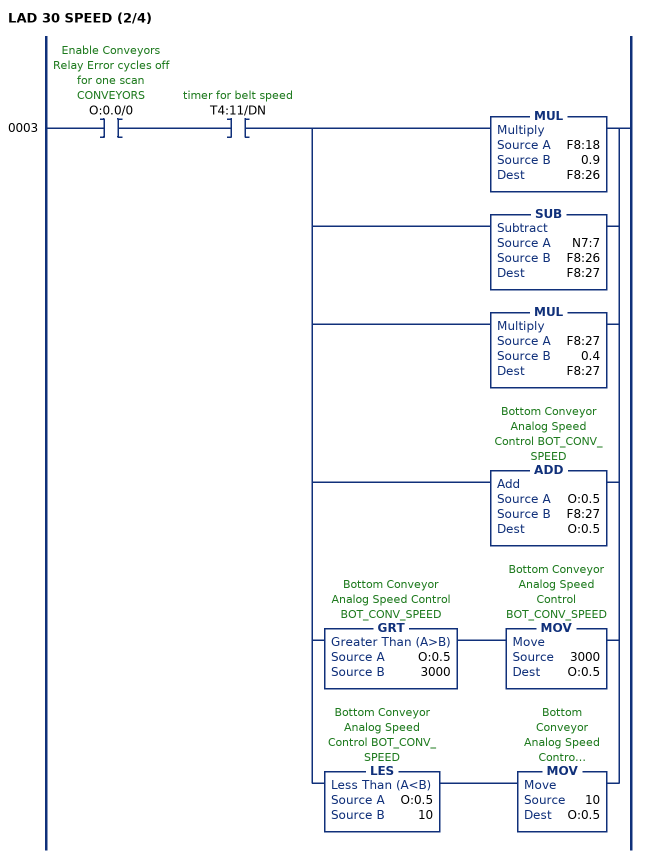
% Rung: 3 %
SOR XIC O:0.0/0 XIC T4:11/DN BST MUL F8:18 0.9 F8:26 NXB SUB N7:7 F8:26 F8:27 NXB MUL F8:27 0.4 F8:27 NXB ADD O:0.5 F8:27 O:0.5 NXB GRT O:0.5 3000 MOV 3000 O:0.5 NXB LES O:0.5 10 MOV 10 O:0.5 BND EOR
%   O:0.0/0  CONVEYORS  "Enable Conveyors Relay Error cycles off for one scan" %
%   T4:11  "timer for belt speed" %
%   F8:18  "top belt speed average in pulses per 100ms" %
%   N7:7  "Top Conv Speed" %
%   O:0.5  BOT_CONV_SPEED  "Bottom Conveyor Analog Speed Control" %

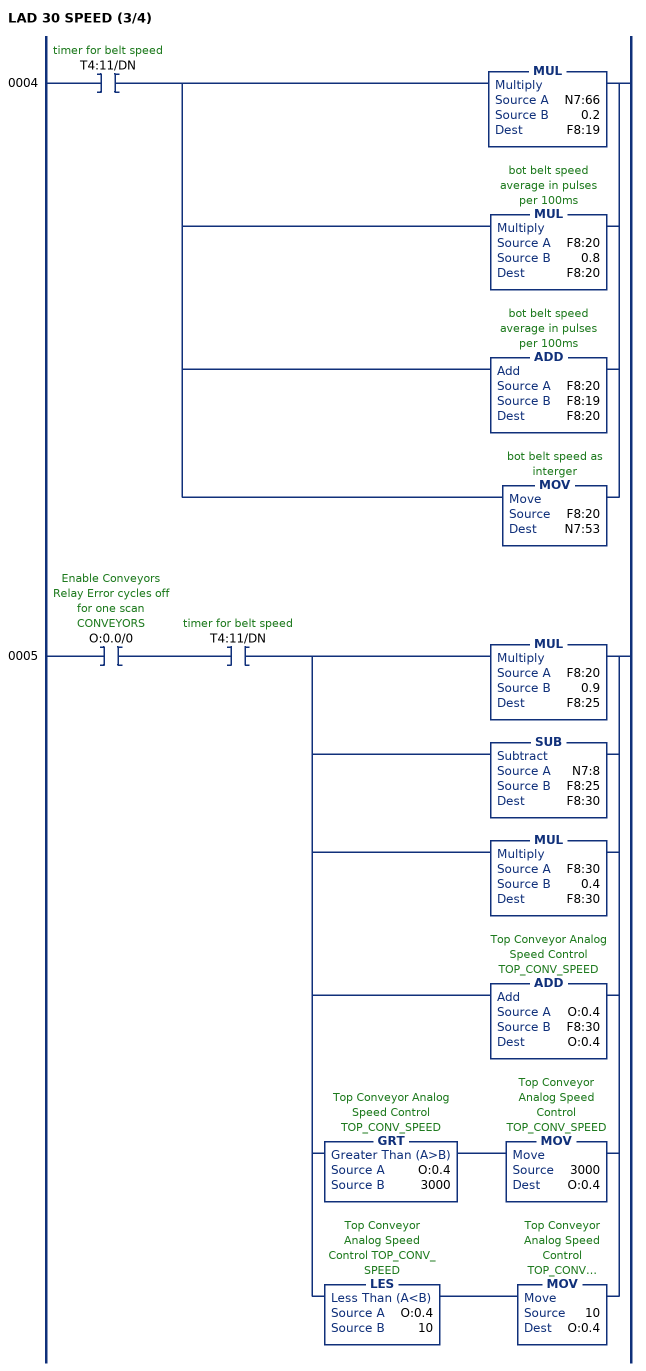
% Rung: 4 %
SOR XIC T4:11/DN BST MUL N7:66 0.2 F8:19 NXB MUL F8:20 0.8 F8:20 NXB ADD F8:20 F8:19 F8:20 NXB MOV F8:20 N7:53 BND EOR
%   T4:11  "timer for belt speed" %
%   N7:66  "pps bottom belt" %
%   F8:20  "bot belt speed average in pulses per 100ms" %
%   N7:53  "bot belt speed as interger" %
% Rung: 5 %
SOR XIC O:0.0/0 XIC T4:11/DN BST MUL F8:20 0.9 F8:25 NXB SUB N7:8 F8:25 F8:30 NXB MUL F8:30 0.4 F8:30 NXB ADD O:0.4 F8:30 O:0.4 NXB GRT O:0.4 3000 MOV 3000 O:0.4 NXB LES O:0.4 10 MOV 10 O:0.4 BND EOR
%   O:0.0/0  CONVEYORS  "Enable Conveyors Relay Error cycles off for one scan" %
%   T4:11  "timer for belt speed" %
%   F8:20  "bot belt speed average in pulses per 100ms" %
%   N7:8  "Bottom Conveyor Speed" %
%   O:0.4  TOP_CONV_SPEED  "Top Conveyor Analog Speed Control" %

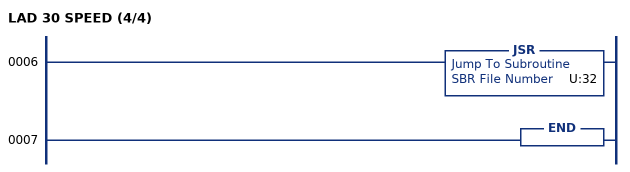
% Rung: 6 %
SOR JSR U:32 EOR
% Rung: 7 %
SOR END EOR

LADDER 32 "BOXER"
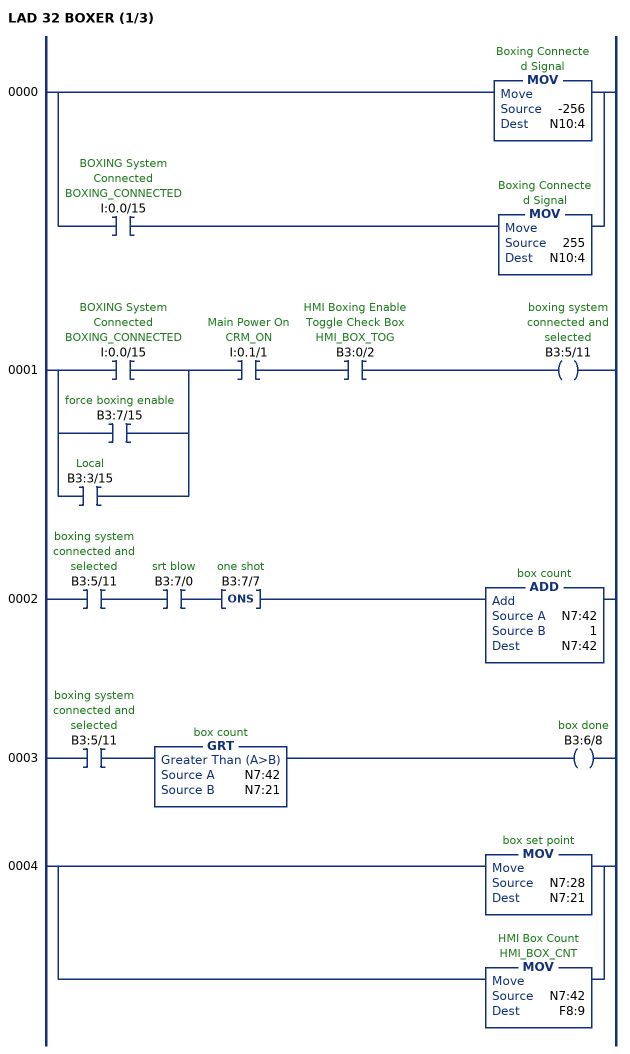
% Rung: 0 %
SOR BST MOV -256 N10:4 NXB XIC I:0.0/15 MOV 255 N10:4 BND EOR
%   N10:4  "Boxing Connected Signal" %
%   I:0.0/15  BOXING_CONNECTED  "BOXING System Connected" %
% Rung: 1 %
SOR BST XIC I:0.0/15 NXB XIC B3:7/15 NXB XIC B3:3/15 BND XIC I:0.1/1 XIC B3:0/2 OTE B3:5/11 EOR
%   I:0.0/15  BOXING_CONNECTED  "BOXING System Connected" %
%   B3:7/15  "force boxing enable" %
%   B3:3/15  "Local" %
%   I:0.1/1  CRM_ON  "Main Power On" %
%   B3:0/2  HMI_BOX_TOG  "HMI Boxing Enable Toggle Check Box" %
%   B3:5/11  "boxing system connected and selected" %
% Rung: 2 %
SOR XIC B3:5/11 XIC B3:7/0 ONS B3:7/7 ADD N7:42 1 N7:42 EOR
%   B3:5/11  "boxing system connected and selected" %
%   B3:7/0  "srt blow" %
%   B3:7/7  "one shot" %
%   N7:42  "box count" %
% Rung: 3 %
SOR XIC B3:5/11 GRT N7:42 N7:21 OTE B3:6/8 EOR
%   B3:5/11  "boxing system connected and selected" %
%   N7:42  "box count" %
%   N7:21  "box set point" %
%   B3:6/8  "box done" %
% Rung: 4 %
SOR BST MOV N7:28 N7:21 NXB MOV N7:42 F8:9 BND EOR
%   N7:28  "box count limit" %
%   N7:21  "box set point" %
%   N7:42  "box count" %
%   F8:9  HMI_BOX_CNT  "HMI Box Count" %

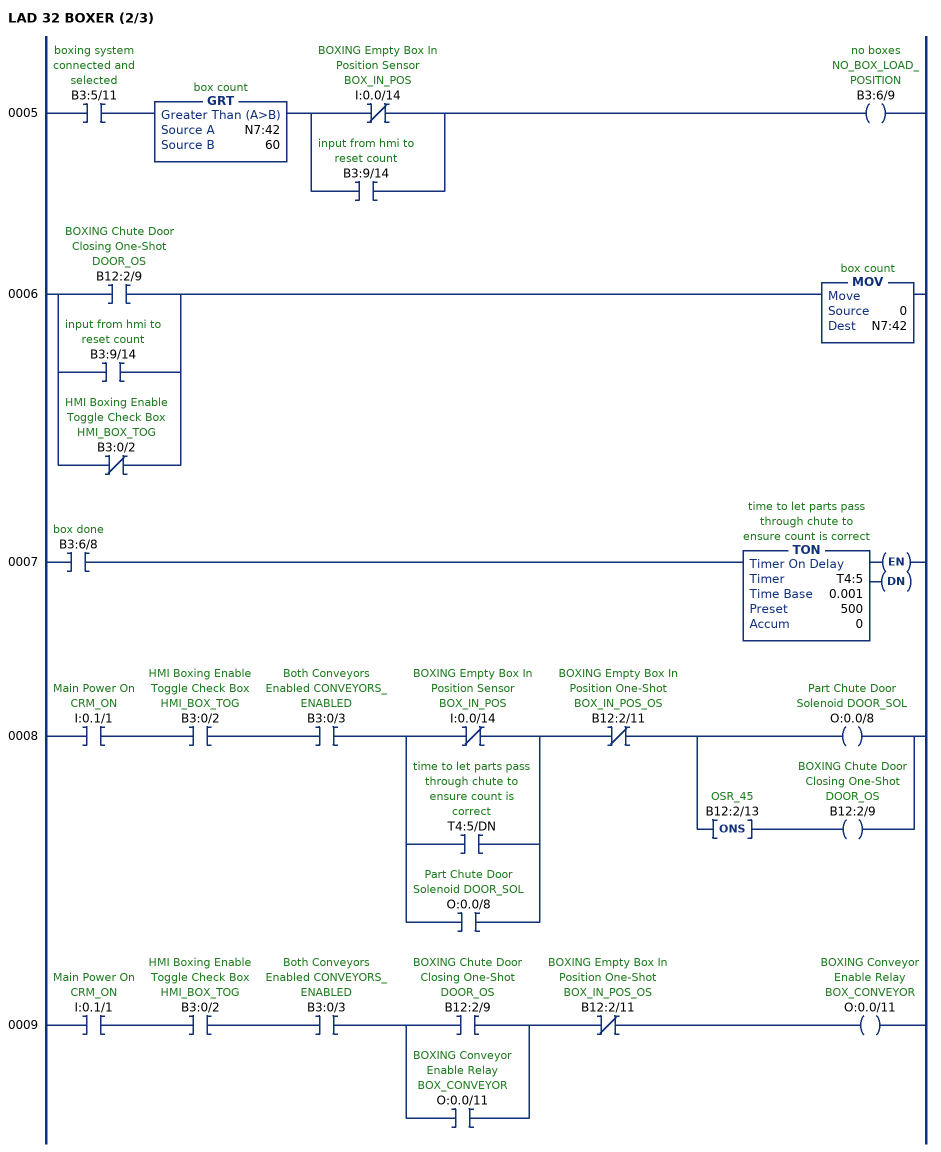
% Rung: 5 %
SOR XIC B3:5/11 GRT N7:42 60 BST XIO I:0.0/14 NXB XIC B3:9/14 BND OTE B3:6/9 EOR
%   B3:5/11  "boxing system connected and selected" %
%   N7:42  "box count" %
%   I:0.0/14  BOX_IN_POS  "BOXING Empty Box In Position Sensor" %
%   B3:9/14  "input from hmi to reset count" %
%   B3:6/9  NO_BOX_LOAD_POSITION  "no boxes" %
% Rung: 6 %
SOR BST XIC B12:2/9 NXB XIC B3:9/14 NXB XIO B3:0/2 BND MOV 0 N7:42 EOR
%   B12:2/9  DOOR_OS  "BOXING Chute Door Closing One-Shot" %
%   B3:9/14  "input from hmi to reset count" %
%   B3:0/2  HMI_BOX_TOG  "HMI Boxing Enable Toggle Check Box" %
%   N7:42  "box count" %
% Rung: 7 %
SOR XIC B3:6/8 TON T4:5 0.001 500 0 EOR
%   B3:6/8  "box done" %
%   T4:5  "time to let parts pass through chute to ensure count is correct" %
% Rung: 8 %
SOR XIC I:0.1/1 XIC B3:0/2 XIC B3:0/3 BST XIO I:0.0/14 NXB XIC T4:5/DN NXB XIC O:0.0/8 BND XIO B12:2/11 BST OTE O:0.0/8 NXB ONS B12:2/13 OTE B12:2/9 BND EOR
%   I:0.1/1  CRM_ON  "Main Power On" %
%   B3:0/2  HMI_BOX_TOG  "HMI Boxing Enable Toggle Check Box" %
%   B3:0/3  CONVEYORS_ENABLED  "Both Conveyors Enabled" %
%   I:0.0/14  BOX_IN_POS  "BOXING Empty Box In Position Sensor" %
%   T4:5  "time to let parts pass through chute to ensure count is correct" %
%   O:0.0/8  DOOR_SOL  "Part Chute Door Solenoid" %
%   B12:2/11  BOX_IN_POS_OS  "BOXING Empty Box In Position One-Shot" %
%   B12:2/13  OSR_45 %
%   B12:2/9  DOOR_OS  "BOXING Chute Door Closing One-Shot" %
% Rung: 9 %
SOR XIC I:0.1/1 XIC B3:0/2 XIC B3:0/3 BST XIC B12:2/9 NXB XIC O:0.0/11 BND XIO B12:2/11 OTE O:0.0/11 EOR
%   I:0.1/1  CRM_ON  "Main Power On" %
%   B3:0/2  HMI_BOX_TOG  "HMI Boxing Enable Toggle Check Box" %
%   B3:0/3  CONVEYORS_ENABLED  "Both Conveyors Enabled" %
%   B12:2/9  DOOR_OS  "BOXING Chute Door Closing One-Shot" %
%   O:0.0/11  BOX_CONVEYOR  "BOXING Conveyor Enable Relay" %
%   B12:2/11  BOX_IN_POS_OS  "BOXING Empty Box In Position One-Shot" %

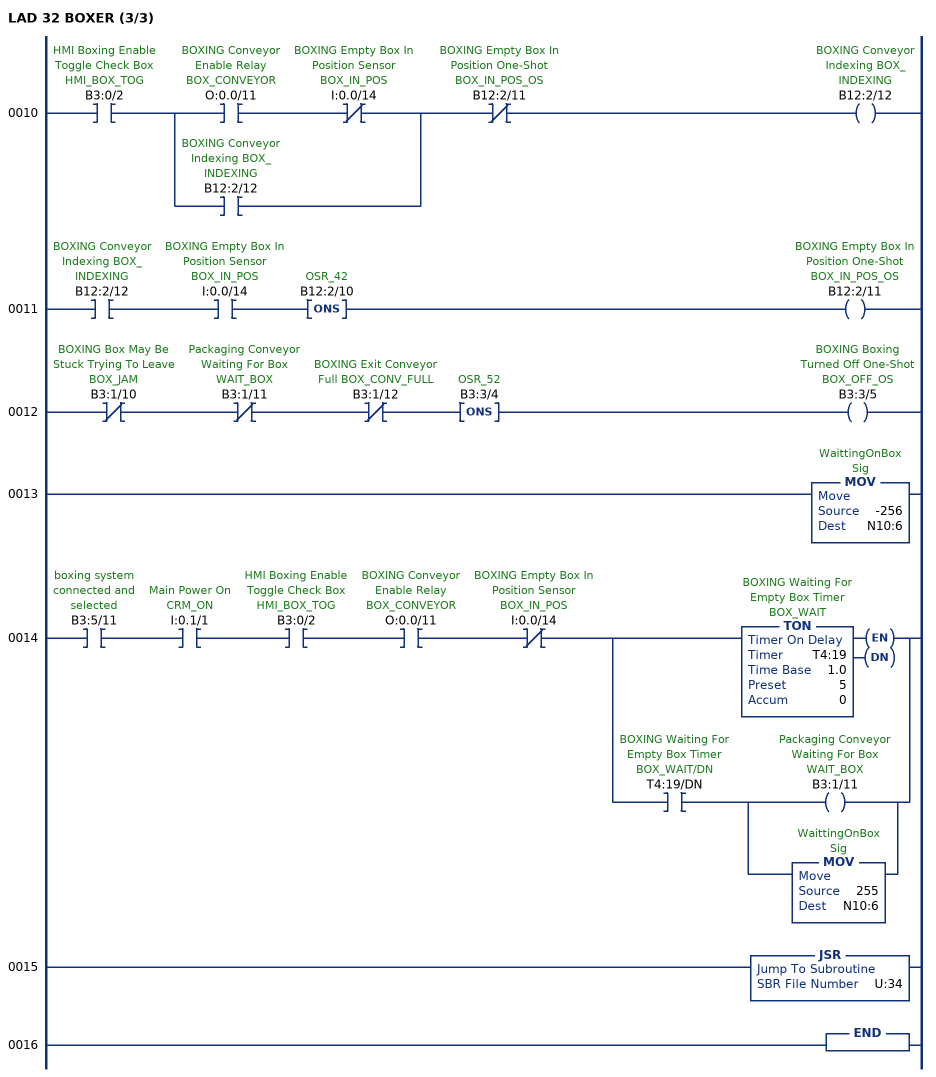
% Rung: 10 %
SOR XIC B3:0/2 BST XIC O:0.0/11 XIO I:0.0/14 NXB XIC B12:2/12 BND XIO B12:2/11 OTE B12:2/12 EOR
%   B3:0/2  HMI_BOX_TOG  "HMI Boxing Enable Toggle Check Box" %
%   O:0.0/11  BOX_CONVEYOR  "BOXING Conveyor Enable Relay" %
%   I:0.0/14  BOX_IN_POS  "BOXING Empty Box In Position Sensor" %
%   B12:2/12  BOX_INDEXING  "BOXING Conveyor Indexing" %
%   B12:2/11  BOX_IN_POS_OS  "BOXING Empty Box In Position One-Shot" %
% Rung: 11 %
SOR XIC B12:2/12 XIC I:0.0/14 ONS B12:2/10 OTE B12:2/11 EOR
%   B12:2/12  BOX_INDEXING  "BOXING Conveyor Indexing" %
%   I:0.0/14  BOX_IN_POS  "BOXING Empty Box In Position Sensor" %
%   B12:2/10  OSR_42 %
%   B12:2/11  BOX_IN_POS_OS  "BOXING Empty Box In Position One-Shot" %
% Rung: 12 %
SOR XIO B3:1/10 XIO B3:1/11 XIO B3:1/12 ONS B3:3/4 OTE B3:3/5 EOR
%   B3:1/10  BOX_JAM  "BOXING Box May Be Stuck Trying To Leave" %
%   B3:1/11  WAIT_BOX  "Packaging Conveyor Waiting For Box" %
%   B3:1/12  BOX_CONV_FULL  "BOXING Exit Conveyor Full" %
%   B3:3/4  OSR_52 %
%   B3:3/5  BOX_OFF_OS  "BOXING Boxing Turned Off One-Shot" %
% Rung: 13 %
SOR MOV -256 N10:6 EOR
%   N10:6  "WaittingOnBoxSig" %
% Rung: 14 %
SOR XIC B3:5/11 XIC I:0.1/1 XIC B3:0/2 XIC O:0.0/11 XIO I:0.0/14 BST TON T4:19 1.0 5 0 NXB XIC T4:19/DN BST OTE B3:1/11 NXB MOV 255 N10:6 BND BND EOR
%   B3:5/11  "boxing system connected and selected" %
%   I:0.1/1  CRM_ON  "Main Power On" %
%   B3:0/2  HMI_BOX_TOG  "HMI Boxing Enable Toggle Check Box" %
%   O:0.0/11  BOX_CONVEYOR  "BOXING Conveyor Enable Relay" %
%   I:0.0/14  BOX_IN_POS  "BOXING Empty Box In Position Sensor" %
%   T4:19  BOX_WAIT  "BOXING Waiting For Empty Box Timer" %
%   B3:1/11  WAIT_BOX  "Packaging Conveyor Waiting For Box" %
%   N10:6  "WaittingOnBoxSig" %
% Rung: 15 %
SOR JSR U:34 EOR
% Rung: 16 %
SOR END EOR

LADDER 34 "CLEANUP"
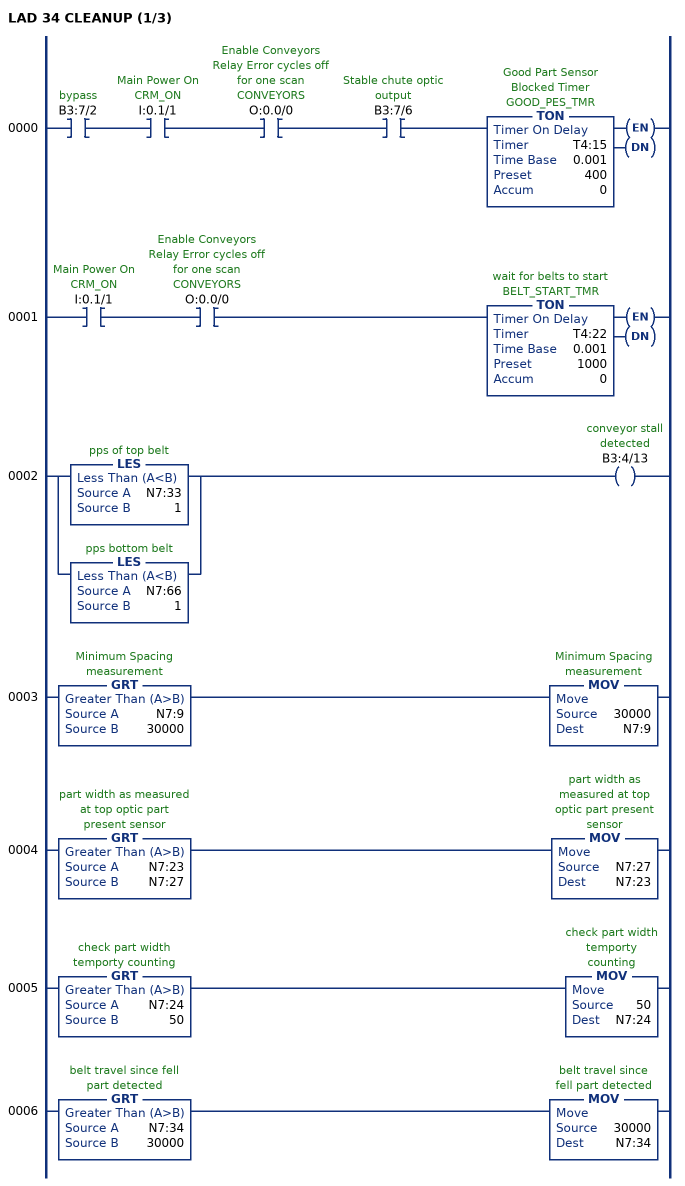
% Rung: 0 %
SOR XIC B3:7/2 XIC I:0.1/1 XIC O:0.0/0 XIC B3:7/6 TON T4:15 0.001 400 0 EOR
%   B3:7/2  "bypass" %
%   I:0.1/1  CRM_ON  "Main Power On" %
%   O:0.0/0  CONVEYORS  "Enable Conveyors Relay Error cycles off for one scan" %
%   B3:7/6  "Stable chute optic output" %
%   T4:15  GOOD_PES_TMR  "Good Part Sensor Blocked Timer" %
% Rung: 1 %
SOR XIC I:0.1/1 XIC O:0.0/0 TON T4:22 0.001 1000 0 EOR
%   I:0.1/1  CRM_ON  "Main Power On" %
%   O:0.0/0  CONVEYORS  "Enable Conveyors Relay Error cycles off for one scan" %
%   T4:22  BELT_START_TMR  "wait for belts to start" %
% Rung: 2 %
SOR BST LES N7:33 1 NXB LES N7:66 1 BND OTE B3:4/13 EOR
%   N7:33  "pps of top belt" %
%   N7:66  "pps bottom belt" %
%   B3:4/13  "conveyor stall detected" %
% Rung: 3 %
SOR GRT N7:9 30000 MOV 30000 N7:9 EOR
%   N7:9  "Minimum Spacing measurement" %
% Rung: 4 %
SOR GRT N7:23 N7:27 MOV N7:27 N7:23 EOR
%   N7:23  "part width as measured at top optic part present sensor" %
%   N7:27  "max part width top optic" %
% Rung: 5 %
SOR GRT N7:24 50 MOV 50 N7:24 EOR
%   N7:24  "check part width temporty counting" %
% Rung: 6 %
SOR GRT N7:34 30000 MOV 30000 N7:34 EOR
%   N7:34  "belt travel since fell part detected" %

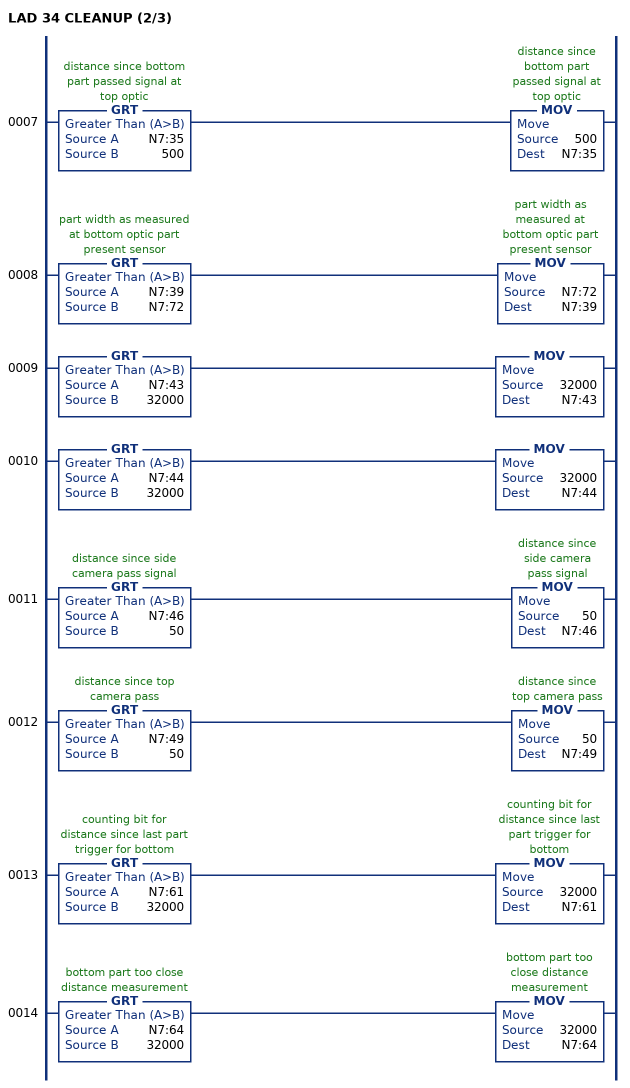
% Rung: 7 %
SOR GRT N7:35 500 MOV 500 N7:35 EOR
%   N7:35  "distance since bottom part passed signal at top optic" %
% Rung: 8 %
SOR GRT N7:39 N7:72 MOV N7:72 N7:39 EOR
%   N7:39  "part width as measured at bottom optic part present sensor" %
%   N7:72  "max part width bottom optic" %
% Rung: 9 %
SOR GRT N7:43 32000 MOV 32000 N7:43 EOR
% Rung: 10 %
SOR GRT N7:44 32000 MOV 32000 N7:44 EOR
% Rung: 11 %
SOR GRT N7:46 50 MOV 50 N7:46 EOR
%   N7:46  "distance since side camera pass signal" %
% Rung: 12 %
SOR GRT N7:49 50 MOV 50 N7:49 EOR
%   N7:49  "distance since top camera pass" %
% Rung: 13 %
SOR GRT N7:61 32000 MOV 32000 N7:61 EOR
%   N7:61  "counting bit for distance since last part trigger for bottom" %
% Rung: 14 %
SOR GRT N7:64 32000 MOV 32000 N7:64 EOR
%   N7:64  "bottom part too close distance measurement" %

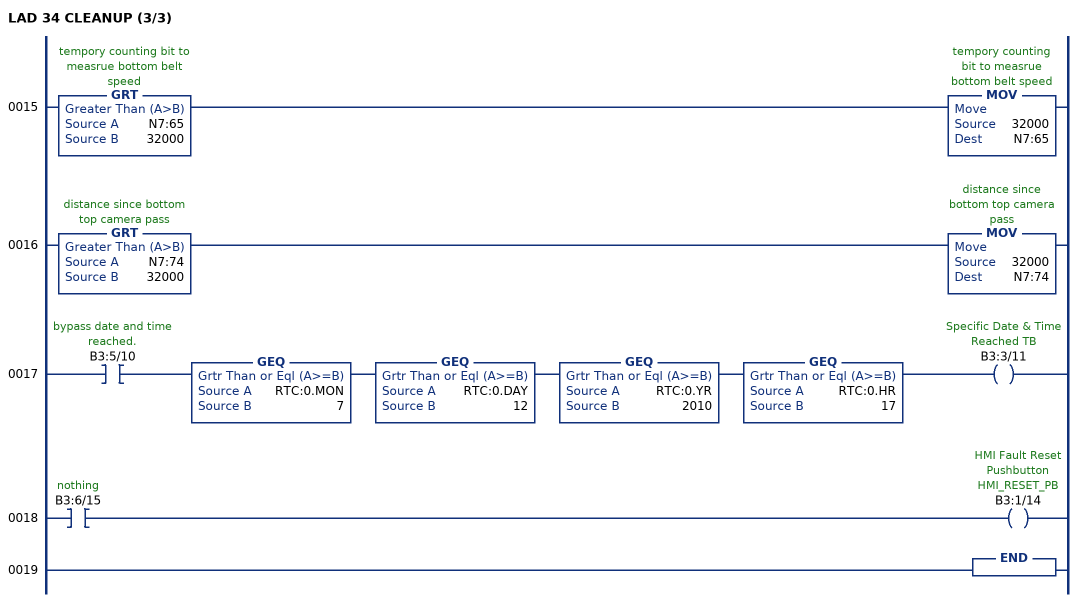
% Rung: 15 %
SOR GRT N7:65 32000 MOV 32000 N7:65 EOR
%   N7:65  "tempory counting bit to measrue bottom belt speed" %
% Rung: 16 %
SOR GRT N7:74 32000 MOV 32000 N7:74 EOR
%   N7:74  "distance since bottom top camera pass" %
% Rung: 17 %
SOR XIC B3:5/10 GEQ RTC:0.MON 7 GEQ RTC:0.DAY 12 GEQ RTC:0.YR 2010 GEQ RTC:0.HR 17 OTE B3:3/11 EOR
%   B3:5/10  "bypass date and time reached." %
%   B3:3/11  TB  "Specific Date & Time Reached" %
% Rung: 18 %
SOR XIC B3:6/15 OTE B3:1/14 EOR
%   B3:6/15  "nothing" %
%   B3:1/14  HMI_RESET_PB  "HMI Fault Reset Pushbutton" %
% Rung: 19 %
SOR END EOR

OTHER DOCUMENTED ADDRESSES
  B3:3/14  "bypass faked part present signal"
  B3:10/14  "Dont use"
  B3:12/0  "Command 1 Oneshot"
  B3:12/1  "Command 1 Active"
  B3:12/2  "Command 2 Oneshot"
  B3:12/3  "Command 2 Active"
  B3:12/4  "Command3 Oneshot"
  B3:12/5  "Command 3 Active"
  B3:12/6  "Inspection Command Counter"
  B3:12/7  "Command 4 Active"
  B3:12/8  "Command 4 Oneshot"
  B3:13/10  "Laser Pass Bit"
  B3:13/11  "Test Spacing From Bottom Camera to Laser"
  B3:13/12  "Test Trigger to laser Spacing"
  B3:13/15  "Test Signals"
  B3:17/12  "Always Off"
  B9:0/0  "Trigger Insert Position"
  B9:0/[N7:2]  "Mask Start Position"
  B9:0/[N7:20]  "part present bit shift load position"
  B9:0/[N17:8]  "part from bottom belt present at top belt optic position"
  B10:0/0  "Pass Insert Position"
  B10:0/1  TOP_CAM_LOAD
  B10:0/[N7:2]  "Pass Bit Position"
  B10:0/[N7:4]  "Pass Insert Position"
  B10:0/[N7:5]  "Pass Start Position"
  B10:0/[N7:6]  "Pass Position"
  B10:0/[N7:48]  TOPCAMTRIGPOS
  B10:0/[N16:4]  "Pass Insert Position"
  B10:0/[N16:6]  "Pass Position"
  B11:0/0  "Trigger Insert Position"
  B11:0/[N7:8]  "Fail Bit Position"
  B11:0/[N16:0]  "Trigger Position"
  B12:1/0  "Conveyor Start Oneshot"
  B12:1/1  "Feed Start Oneshot"
  B12:1/2  "Conveyor Stop Oneshot"
  B12:1/3  "Feed Stop Oneshot"
  B12:1/5  "Conveyor Start Oneshot"
  B12:2/8  BOXING  "BOXING System Wiring Is Connected"
  B12:2/14  BOX_PLC_COUNTER  "BOXING PLC Counter Active Bit"
  B14:0/0  "Bottom Pass Insert"
  B14:0/4  "Bottom Pass Insert Position"
  B14:0/[N13:14]  "Start Laser Pass"
  B14:0/[N16:4]  "Pass Insert Position"
  B14:0/[N16:6]  "Pass Position"
  B15:0  "Alarm Bits"
  B18:1/1  "bottom pass one shot transfer"
  B18:3/2  "Part Present Oneshot"
  B18:3/3  "Part Present Oneshot"
  B18:142  "fack camerea pass signal"
  B22:0  "Transfer Shift Register"
  B22:0/0  "load top conveyor bitshift from bottom cammera pass."
  B22:0/[N17:8]  "bottom good part at top optic position"
  B23:0/[N7:0]  "Bottom Pass Output"
  B25:0/4  UNUSED_4  "Unused Camera #4 Trigger"
  C5:2  "Fault Counter"
  C5:5  "Trigger Count"
  C5:6  "Trigger Counter"
  C5:7  "Complete Counter"
  C5:8  BOX_CNT_1  "BOXING Quantity Counter #1"
  C5:9  BOX_CNT_2  "BOXING Quantity Counter #1"
  F19:0  BOT_HS_COUNTER  "Bottom Encoder High Speed Counter"
  F19:4  "Conveyor Input Blip Counter"
  HSC:0  "top conveyor"
  HSC:1  "bottom conveyor"
  I:0.0/1  "Part Counter P.E."
  I:0.0/7  PYRAMID_PASS  "VISION SYSTEM Inspection Complete"
  I:0.0/11  "Conveyor Start"
  I:0.1/2  BOT_TRIGGER_PES  "Bottom Conveyor Part Trigger Sensor"
  N7:78  "Top Belt Speed As interger"
  N13:0  "Part Inspecting"
  N13:4  "Completed Counter"
  N13:5  "Trigger Position Counter"
  N13:6  "BlowOff Start Counter"
  N13:7  "BlowOff Stop Counter"
  N13:8  "Inspection Command Counter"
  N13:9  "Complete Counter"
  N13:10  "Pass Signal Counter"
  N13:11  "Solenoid Signal Counter"
  N13:12  "Hold Pass Counter"
  N13:13  "Hold Pass Length"
  N16:1  "Bottom Inspection Offset For Tracking"
  N16:3  "Bit Shift Preset"
  N17:5  "Parts In Tube Counter"
  N17:6  "Parts In Tube Limit"
  N17:9  "Bot to Top Transfer Position"
  N17:12  "Trigger to laser Counter"
  O:0.0/1  TOP_RINGLIGHT  "Camera "F" Top View Ringlight Enable"
  PFILE:6  "check for part jams"
  R6:5.POS  "Empty Fifo"
  T23:0  T25

COMMENTS NOT ATTACHED TO A CURRENT RUNG
  F8:13: *************************
    Loads Side Camera Passing data into a bit shift
    *************************
    
    loads passing data bit into passing data bit shift register at the part present cl.
  I:0.0/8: special rung for testing. This rung can simulate a pass signal. It will not be timed correctly.
  B23:0/0: Yet another bit shift load with data in the part position indicating that there was a bottom system part pass as well as a top system part present at this location.
    
    verified works w/bypassed 071910 and unbypassed 072010
  I:0.0/6: In this rung I'm adding the capibility to fake a bottom camera pass signal for testing purpouspes.
  C5:4: tempory counting to verify pass part count with boxing part count.
  B22:0/0: ***********************
     Bottom Part Syncronizing Logic
    ***********************
    
    This is the point at the bottom of the top conveyor where the part jumps from the bottom conveyor.  This system will then track the part through the top system to the point of the laser optic in order to verify that the part in question has passed the bottom inspection.  I believe that we NEED to include FAILING inspections to eliminate the possibility of a out of position part from passing. LW 072010
  T20:2.ACC: This rung is starting a timer that should be activated directly before the laser optic part presense sensor on the top conveyer and should cause the top optic to be ignored if the bottom camera system didn't pass. however other arrangements must be made if the bottom camera isn't going to be used as is the case with a nut inspection.
  T20:2: The timer used to verify that the part that triggered the top laser optic has passed the bottom camer. needs to be count
  N17:8: ****************************************************************************************************************
    I can not find anywhere in the program where the "Test Spacing From Pickup to Trigger is activated indicating to me that this entire function must not be doing anything in this program at this time.
    ****************************************************************************************************************
  B11:0/0: load part present bit shit with one shot data from the part present sensor
  B3:7/9: ************************************
     The next 3 rungs appear to do nothing
    ***********************************
  T4:0: **************
    Side Camera Trigger
    *************
    
    Trigger top camera (side)
  F8:0: Counter inside of a high speed counter interrupt counts the number of Bit Shifts that need to be processed in order to move the logic with the parts on the conveyor.
  N7:45: not fully functional because of part overlap but measurems the camera responce time when part inspections are not overlaping
  F19:0: Counter inside of a high speed counter interrupt counts the number of Bit Shifts that need to be processed in order to move the logic with the parts on the conveyor.
  F8:14: **************
    Bottom Top Camera Trigger
    *************
    
    Trigger Bottom Top Camera

DATA TABLE (non-zero values as saved)
DATA B3
% B3:0 % 0X0010 0X0100 0X0000 0X4014 0X2C01 0X6280 0X4049 0X0026 0X0000 0X8000
% B3:10 % 0X2070
DATA T4
% .PRE .ACC %
% T4:0 % 5 0
% T4:1 % 5 0
% T4:2 % 20 0
% T4:3 % 1000 0
% T4:4 % 100 0
% T4:5 % 500 0
% T4:6 % 900 0
% T4:7 % 1000 0
% T4:8 % 1000 0
% T4:9 % 16 0
% T4:10 % 5000 5001
% T4:11 % 500 183
% T4:12 % 10 0
% T4:13 % 999 0
% T4:14 % 999 0
% T4:15 % 400 0
% T4:16 % 999 0
% T4:17 % 1000 0
% T4:18 % 5 0
% T4:19 % 5 0
% T4:20 % 10 0
% T4:21 % 6 0
% T4:22 % 1000 0
% T4:23 % 1000 0
% T4:24 % 1000 0
% T4:25 % 20 9
DATA R6
% .LEN .POS %
% R6:0 % 1600 0
% R6:1 % 600 0
% R6:2 % 1600 0
DATA N7
% N7:0 % 794 20 4 885 170 46 1106 100 100 0
% N7:10 % 1 0 0 0 20 0 30 746 45 15
% N7:20 % 0 20300 0 0 0 85 -398 12 20300 650
% N7:30 % 0 716 716 0 651 0 30 0 0 0
% N7:40 % 1253 300 0 32000 32000 0 50 794 801 50
% N7:50 % 801 113 5959 0 126 0 0 0 983 0
% N7:60 % 1 0 0 15 0 0 0 0 0 0
% N7:70 % 0 0 15 0 32000 0 185 0 12 0
% N7:80 % 0 170 4 50 9999 0 0 0 0 0
DATA F8
% F8:0 % 1.512617e+07 1.677722e+07 1.419693e+07 1.677722e+07 1174317
% F8:5 % 640628 1.677722e+07 1445642 8097655 0
% F8:10 % 600 0.093 914 5 200
% F8:15 % 12000 5958.514 0 0 0
% F8:20 % 0 0 1.13 0 0
% F8:25 % 99.67899 99.90447 0.03821106 1.677722e+07 1.677722e+07
% F8:30 % 0.1284027 0 0 0 0
DATA B9
% B9:100 % 0X0000 0X0000 0X0100 0X0000 0X0400 0X0000 0X0002 0X0000 0X0000 0X0000
% B9:110 % 0X0000 0X0000 0X0000 0X0000 0X0010 0X0000 0X0000 0X0000 0X0000 0X0000
% B9:120 % 0X0000 0X0000 0X0400 0X0000 0X0000 0X8800 0X0000 0X0000 0X0000 0X0000
% B9:130 % 0X0000 0X0000 0X0000 0X0000 0X2000 0X0000 0X0000 0X0000 0X0000 0X8000
% B9:140 % 0X2480 0X0000 0X0000 0X0000 0X0000 0X0000 0X0000 0X0000 0X0000 0X0000
% B9:160 % 0X0000 0X0000 0X0000 0X0000 0X0000 0X0000 0X2000 0X0002 0X0000 0X0000
% B9:170 % 0X0000 0X0000 0X0000 0X2000 0X0000 0X0000 0X0000 0X0000 0X0000 0X0000
% B9:180 % 0X0000 0X0000 0X0000 0X0000 0X0000 0X0002 0X0000 0X0000 0X0000 0X0000
% B9:190 % 0X0010 0X0000 0X0000 0X0000 0X0000 0X0000 0X0000 0X0000 0X0000 0X0000
% B9:200 % 0X0000 0X0000 0X0000 0X0010 0X0000 0X2000 0X0000 0X0000 0X0000 0X0000
% B9:220 % 0X0000 0X0000 0X0000 0X0200 0X0000 0X0000 0X0000 0X0000 0X0000 0X0020
% B9:230 % 0X0040 0X0000 0X0000 0X0000 0X0000 0X0000 0X0000 0X0000 0X0000 0X0000
DATA N10
% N10:0 % -256 -256 -256 -256 255 -256 -256 -256 -256 -256
% N10:10 % -256 -256 -256 0 0 0 0 0 0 0
DATA B11
% B11:180 % 0X0000 0X8000 0X0000 0X0000 0X0000 0X0000 0X0000 0X0000 0X0000 0X0000
% B11:240 % 0X0000 0X0000 0X0000 0X4000 0X0000 0X0000 0X0000 0X0000 0X0000 0X0000
DATA B12
% B12:0 % 0X0000 0X000C 0X0100
DATA N16
% N16:0 % 85
DATA T20
% .PRE .ACC %
% T20:0 % 5 0
DATA R21
% .LEN .POS %
% R21:0 % 1300 0
% R21:1 % 1000 0
% R21:2 % 1300 0
% R21:3 % 1000 0
